// TIA Portal V19 export
DATA_BLOCK "IO-LinkDeviceEventData"   // DB211
{ S7_Optimized_Access := 'TRUE' }
// 10 Bytes per device
// stored: AutoNumber false, MemoryReserve 0
   VAR RETAIN
      V0930 : "_EV_DataUDT";
      V0931 : "_EV_DataUDT";
      V0552 : "_EV_DataUDT";
      V0934 : "_EV_DataUDT";
      V0935 : "_EV_DataUDT";
      V0940 : "_EV_DataUDT";
      V0941 : "_EV_DataUDT";
      V0942 : "_EV_DataUDT";
      V0943 : "_EV_DataUDT";
      V0944 : "_EV_DataUDT";
      AL2221_100_005_X06 : "_EV_DataUDT";
      V1021 : "_EV_DataUDT";
      V1023 : "_EV_DataUDT";
      V1024 : "_EV_DataUDT";
      V1025 : "_EV_DataUDT";
      V1027 : "_EV_DataUDT";
      V1083 : "_EV_DataUDT";
      V0936 : "_EV_DataUDT";
   END_VAR
BEGIN
END_DATA_BLOCK
